(* IEC 61131-3 sources: IRIS-Project/LASAL CONTROL SOFTWARE/LasalProject_2025_09_12/Class/IrrTimerManager, 1 file *)

(* ---- IrrTimerManager.st ---- *)
(*!
<Class
	Name               = "IrrTimerManager"
	Revision           = "0.0"
	RealtimeTask       = "false"
	CyclicTask         = "false"
	BackgroundTask     = "false"
	Sigmatek           = "false"
	OSInterface        = "false"
	HighPriority       = "false"
	Automatic          = "false"
	UpdateMode         = "Prescan"
	SharedCommandTable = "true"
	Objectsize         = "(358,120)">
	<Channels>
		<Server Name="ClassSvr" Visualized="false" Initialize="false" WriteProtected="true" Retentive="false"/>
		<Client Name="NrIrrTablets" Required="true" Internal="false"/>
		<Client Name="SetStartStopIrr" Required="true" Internal="false"/>
		<Client Name="TabletInIrrPos" Required="true" Internal="false"/>
		<Client Name="TimerManager2" Required="true" Internal="true"/>
	</Channels>
	<Network Name="IrrTimerManager">
		<!-- List of Components in this network -->
		<Components>
			<Object
				Name       = "TimerManager2"
				Class      = "IrradiationManager"
				Position   = "(1230,210)"
				Visualized = "false"
				CyclicTime = "100 ms">
				<Channels>
					<Server Name="ClassSvr"/>
					<Server Name="s_1_3_pelletMode"/>
					<Server Name="s_EasyGUI"/>
					<Server Name="s_Reset"/>
					<Server Name="s_setTimer1"/>
					<Server Name="s_setTimer2"/>
					<Server Name="s_setTimer3"/>
					<Server Name="s_TimerStartStop"/>
					<Server Name="s_VisTimerIrr1"/>
					<Server Name="s_VisTimerIrr2"/>
					<Server Name="s_VisTimerIrr3"/>
					<Server Name="s_VisTimerIrrAdv1"/>
					<Server Name="s_VisTimerIrrAdv2"/>
					<Server Name="s_VisTimerIrrAdv3"/>
					<Server Name="Startprocess"/>
					<Client Name="c_SysTime"/>
					<Client Name="c_timerLib"/>
					<Client Name="NrIrrTablets"/>
					<Client Name="SetStartStopIrr"/>
					<Client Name="TabletInIrrPos"/>
					<Client Name="Timer1"/>
					<Client Name="Timer2"/>
					<Client Name="Timer3"/>
				</Channels>
			</Object>
		</Components>
		<Comments>
		</Comments>
		<!-- List of Connections in this network -->
		<Connections>
			<Connection Source="this.TimerManager2" Destination="TimerManager2.ClassSvr"/>
			<Connection Source="TimerManager2.TabletInIrrPos" Destination="this.TabletInIrrPos" Vertices="(1230,540),(330,630),(330,210),(38,210),"/>
			<Connection Source="TimerManager2.NrIrrTablets" Destination="this.NrIrrTablets" Vertices="(1230,600),(300,660),(300,270),(38,270),"/>
			<Connection Source="TimerManager2.SetStartStopIrr" Destination="this.SetStartStopIrr" Vertices="(1230,720),(270,720),(270,330),(38,330),"/>
		</Connections>
		<!-- Headerfiles -->
		<Options>
		</Options>
	</Network>
</Class>
*)
IrrTimerManager : CLASS
  //Servers:
	ClassSvr 	: SvrChCmd_DINT;
  //Clients:
	TabletInIrrPos 	: CltCh_DINT;
	NrIrrTablets 	: CltCh_DINT;
	SetStartStopIrr 	: CltCh_t_IrradiationPhase_PTofCls_Manager_globale;
	TimerManager2 	: CltChCmd_IrradiationManager;
  //Variables:
  //Functions:
  //Tables:
	FUNCTION @STD
		VAR_OUTPUT
			ret_code	: CONFSTATES;
		END_VAR;
	FUNCTION GLOBAL TAB @CT_;
END_CLASS;

#pragma using IrradiationManager
